FUNCTION_BLOCK FB_MatrixInvert_Test EXTENDS FB_TestSuite
VAR_INPUT
END_VAR
VAR_OUTPUT
END_VAR
VAR
END_VAR

WhenIdentityExpectIdentity();
WhenSingularExpectError();
WhenSolvableExpectSolution();

METHOD PRIVATE WhenIdentityExpectIdentity
VAR_INPUT
END_VAR
VAR
	M1 : DynamicMatrix;
	M2 : DynamicMatrix;
	Result : BOOL;
END_VAR
TEST('WhenIdentityExpectIdentity');

// @TEST-RUN
M1.InitIdentity(3);
M2.InitIdentity(3);
Result := M2.InvertSquare(1E-9);

// @TEST-ASSERT
AssertTrue(Result,'Main function call was not successful');
AssertTrue(M1.IsNearlyEqual(M2,1E-6),'Result was not the same');

TEST_FINISHED();
END_METHOD

METHOD PRIVATE WhenSingularExpectError
VAR_INPUT
END_VAR
VAR
	M1 : DynamicMatrix;
	M2 : DynamicMatrix;
	Result : BOOL;
END_VAR
TEST('WhenSingularExpectError');

// @TEST-RUN
M1.InitTrapezoidal(3,3,1,1,1);
Result := M2.AsInverse(M1,1E-9);

// @TEST-ASSERT
AssertFalse(Result,'Main function call was surprisingly successful');

TEST_FINISHED();
END_METHOD

METHOD PRIVATE WhenSolvableExpectSolution
VAR_INPUT
END_VAR
VAR
	M1 : DynamicMatrix;
	M2 : DynamicMatrix;
	M3 : DynamicMatrix;
	M4 : DynamicMatrix;
	Result : BOOL;
END_VAR
TEST('WhenSolvableExpectSolution');

// @TEST-RUN
M1.InitIdentity(3);
M2.InitMagicSquare(3);
Result := M3.AsInverse(M2,1E-9);
M4.AsMatrixProduct(M2,M3);

// @TEST-ASSERT
AssertTrue(Result,'Main function call was not successful');
AssertTrue(M1.IsNearlyEqual(M4,1E-6),'Result was not a true inverse');

TEST_FINISHED();
END_METHOD

END_FUNCTION_BLOCK

(* stored: Version 1.1.0.1, ProductVersion 3.1.4024.9
   POU FB_MatrixInvert_Test: Id {58e64662-6852-0ee1-3386-4bd0e41d7b01}, SpecialFunc None
   Method WhenIdentityExpectIdentity: Id {78d2eada-d22c-013f-2c4c-82c721cf973f}
   Method WhenSingularExpectError: Id {4b469611-5b6d-0dd5-3f12-a06b3d86ec57}
   Method WhenSolvableExpectSolution: Id {99550ef7-96d5-0f67-03af-0b05c32633ba} *)
